FUNCTION_BLOCK E_MERGE (* Merge(OR)of multiple events *)
  (* Standard: 61499-2 *)
  (* Version 0.2, 2008-07-02, JHC, Holobloc Inc, Corrected package in header. *)
  (* Version 0.1, 2000-10-18, JHC, Rockwell Automation, XML version *)
  (* Version 0.0, 1998-11-19, JHC, Rockwell Automation, SRC version *)
  (* Compiler header: package fb.rt.events; *)
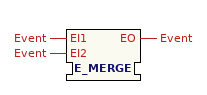
  EVENT_INPUT
    EI1; (* First input event *)
    EI2; (* Second input event *)
  END_EVENT
  EVENT_OUTPUT
    EO; (* Output Event *)
  END_EVENT
END_FUNCTION_BLOCK
